   // GBK_TO_UNICODE[42068] := 16#F758;
   // GBK_TO_UNICODE[42069] := 16#9C54;
   // GBK_TO_UNICODE[42070] := 16#F759;
   // GBK_TO_UNICODE[42071] := 16#9C55;
   // GBK_TO_UNICODE[42072] := 16#F75A;
   // GBK_TO_UNICODE[42073] := 16#9C56;
   // GBK_TO_UNICODE[42074] := 16#F75B;
   // GBK_TO_UNICODE[42075] := 16#9C57;
   // GBK_TO_UNICODE[42076] := 16#F75C;
   // GBK_TO_UNICODE[42077] := 16#9C58;
   // GBK_TO_UNICODE[42078] := 16#F75D;
   // GBK_TO_UNICODE[42079] := 16#9C59;
   // GBK_TO_UNICODE[42080] := 16#F75E;
   // GBK_TO_UNICODE[42081] := 16#9C5A;
   // GBK_TO_UNICODE[42082] := 16#F75F;
   // GBK_TO_UNICODE[42083] := 16#9C5B;
   // GBK_TO_UNICODE[42084] := 16#F760;
   // GBK_TO_UNICODE[42085] := 16#9C5C;
   // GBK_TO_UNICODE[42086] := 16#F761;
   // GBK_TO_UNICODE[42087] := 16#9C5D;
   // GBK_TO_UNICODE[42088] := 16#F762;
   // GBK_TO_UNICODE[42089] := 16#9C5E;
   // GBK_TO_UNICODE[42090] := 16#F763;
   // GBK_TO_UNICODE[42091] := 16#9C5F;
   // GBK_TO_UNICODE[42092] := 16#F764;
   // GBK_TO_UNICODE[42093] := 16#9C60;
   // GBK_TO_UNICODE[42094] := 16#F765;
   // GBK_TO_UNICODE[42095] := 16#9C61;
   // GBK_TO_UNICODE[42096] := 16#F766;
   // GBK_TO_UNICODE[42097] := 16#9C62;
   // GBK_TO_UNICODE[42098] := 16#F767;
   // GBK_TO_UNICODE[42099] := 16#9C63;
   // GBK_TO_UNICODE[42100] := 16#F768;
   // GBK_TO_UNICODE[42101] := 16#9C64;
   // GBK_TO_UNICODE[42102] := 16#F769;
   // GBK_TO_UNICODE[42103] := 16#9C65;
   // GBK_TO_UNICODE[42104] := 16#F76A;
   // GBK_TO_UNICODE[42105] := 16#9C66;
   // GBK_TO_UNICODE[42106] := 16#F76B;
   // GBK_TO_UNICODE[42107] := 16#9C67;
   // GBK_TO_UNICODE[42108] := 16#F76C;
   // GBK_TO_UNICODE[42109] := 16#9C68;
   // GBK_TO_UNICODE[42110] := 16#F76D;
   // GBK_TO_UNICODE[42111] := 16#9C69;
   // GBK_TO_UNICODE[42112] := 16#F76E;
   // GBK_TO_UNICODE[42113] := 16#9C6A;
   // GBK_TO_UNICODE[42114] := 16#F76F;
   // GBK_TO_UNICODE[42115] := 16#9C6B;
   // GBK_TO_UNICODE[42116] := 16#F770;
   // GBK_TO_UNICODE[42117] := 16#9C6C;
   // GBK_TO_UNICODE[42118] := 16#F771;
   // GBK_TO_UNICODE[42119] := 16#9C6D;
   // GBK_TO_UNICODE[42120] := 16#F772;
   // GBK_TO_UNICODE[42121] := 16#9C6E;
   // GBK_TO_UNICODE[42122] := 16#F773;
   // GBK_TO_UNICODE[42123] := 16#9C6F;
   // GBK_TO_UNICODE[42124] := 16#F774;
   // GBK_TO_UNICODE[42125] := 16#9C70;
   // GBK_TO_UNICODE[42126] := 16#F775;
   // GBK_TO_UNICODE[42127] := 16#9C71;
   // GBK_TO_UNICODE[42128] := 16#F776;
   // GBK_TO_UNICODE[42129] := 16#9C72;
   // GBK_TO_UNICODE[42130] := 16#F777;
   // GBK_TO_UNICODE[42131] := 16#9C73;
   // GBK_TO_UNICODE[42132] := 16#F778;
   // GBK_TO_UNICODE[42133] := 16#9C74;
   // GBK_TO_UNICODE[42134] := 16#F779;
   // GBK_TO_UNICODE[42135] := 16#9C75;
   // GBK_TO_UNICODE[42136] := 16#F77A;
   // GBK_TO_UNICODE[42137] := 16#9C76;
   // GBK_TO_UNICODE[42138] := 16#F77B;
   // GBK_TO_UNICODE[42139] := 16#9C77;
   // GBK_TO_UNICODE[42140] := 16#F77C;
   // GBK_TO_UNICODE[42141] := 16#9C78;
   // GBK_TO_UNICODE[42142] := 16#F77D;
   // GBK_TO_UNICODE[42143] := 16#9C79;
   // GBK_TO_UNICODE[42144] := 16#F77E;
   // GBK_TO_UNICODE[42145] := 16#9C7A;
   // GBK_TO_UNICODE[42146] := 16#F780;
   // GBK_TO_UNICODE[42147] := 16#9C7B;
   // GBK_TO_UNICODE[42148] := 16#F781;
   // GBK_TO_UNICODE[42149] := 16#9C7D;
   // GBK_TO_UNICODE[42150] := 16#F782;
   // GBK_TO_UNICODE[42151] := 16#9C7E;
   // GBK_TO_UNICODE[42152] := 16#F783;
   // GBK_TO_UNICODE[42153] := 16#9C80;
   // GBK_TO_UNICODE[42154] := 16#F784;
   // GBK_TO_UNICODE[42155] := 16#9C83;
   // GBK_TO_UNICODE[42156] := 16#F785;
   // GBK_TO_UNICODE[42157] := 16#9C84;
   // GBK_TO_UNICODE[42158] := 16#F786;
   // GBK_TO_UNICODE[42159] := 16#9C89;
   // GBK_TO_UNICODE[42160] := 16#F787;
   // GBK_TO_UNICODE[42161] := 16#9C8A;
   // GBK_TO_UNICODE[42162] := 16#F788;
   // GBK_TO_UNICODE[42163] := 16#9C8C;
   // GBK_TO_UNICODE[42164] := 16#F789;
   // GBK_TO_UNICODE[42165] := 16#9C8F;
   // GBK_TO_UNICODE[42166] := 16#F78A;
   // GBK_TO_UNICODE[42167] := 16#9C93;
   // GBK_TO_UNICODE[42168] := 16#F78B;
   // GBK_TO_UNICODE[42169] := 16#9C96;
   // GBK_TO_UNICODE[42170] := 16#F78C;
   // GBK_TO_UNICODE[42171] := 16#9C97;
   // GBK_TO_UNICODE[42172] := 16#F78D;
   // GBK_TO_UNICODE[42173] := 16#9C98;
   // GBK_TO_UNICODE[42174] := 16#F78E;
   // GBK_TO_UNICODE[42175] := 16#9C99;
   // GBK_TO_UNICODE[42176] := 16#F78F;
   // GBK_TO_UNICODE[42177] := 16#9C9D;
   // GBK_TO_UNICODE[42178] := 16#F790;
   // GBK_TO_UNICODE[42179] := 16#9CAA;
   // GBK_TO_UNICODE[42180] := 16#F791;
   // GBK_TO_UNICODE[42181] := 16#9CAC;
   // GBK_TO_UNICODE[42182] := 16#F792;
   // GBK_TO_UNICODE[42183] := 16#9CAF;
   // GBK_TO_UNICODE[42184] := 16#F793;
   // GBK_TO_UNICODE[42185] := 16#9CB9;
   // GBK_TO_UNICODE[42186] := 16#F794;
   // GBK_TO_UNICODE[42187] := 16#9CBE;
   // GBK_TO_UNICODE[42188] := 16#F795;
   // GBK_TO_UNICODE[42189] := 16#9CBF;
   // GBK_TO_UNICODE[42190] := 16#F796;
   // GBK_TO_UNICODE[42191] := 16#9CC0;
   // GBK_TO_UNICODE[42192] := 16#F797;
   // GBK_TO_UNICODE[42193] := 16#9CC1;
   // GBK_TO_UNICODE[42194] := 16#F798;
   // GBK_TO_UNICODE[42195] := 16#9CC2;
   // GBK_TO_UNICODE[42196] := 16#F799;
   // GBK_TO_UNICODE[42197] := 16#9CC8;
   // GBK_TO_UNICODE[42198] := 16#F79A;
   // GBK_TO_UNICODE[42199] := 16#9CC9;
   // GBK_TO_UNICODE[42200] := 16#F79B;
   // GBK_TO_UNICODE[42201] := 16#9CD1;
   // GBK_TO_UNICODE[42202] := 16#F79C;
   // GBK_TO_UNICODE[42203] := 16#9CD2;
   // GBK_TO_UNICODE[42204] := 16#F79D;
   // GBK_TO_UNICODE[42205] := 16#9CDA;
   // GBK_TO_UNICODE[42206] := 16#F79E;
   // GBK_TO_UNICODE[42207] := 16#9CDB;
   // GBK_TO_UNICODE[42208] := 16#F79F;
   // GBK_TO_UNICODE[42209] := 16#9CE0;
   // GBK_TO_UNICODE[42210] := 16#F7A0;
   // GBK_TO_UNICODE[42211] := 16#9CE1;
   // GBK_TO_UNICODE[42212] := 16#F7A1;
   // GBK_TO_UNICODE[42213] := 16#9CCC;
   // GBK_TO_UNICODE[42214] := 16#F7A2;
   // GBK_TO_UNICODE[42215] := 16#9CCD;
   // GBK_TO_UNICODE[42216] := 16#F7A3;
   // GBK_TO_UNICODE[42217] := 16#9CCE;
   // GBK_TO_UNICODE[42218] := 16#F7A4;
   // GBK_TO_UNICODE[42219] := 16#9CCF;
   // GBK_TO_UNICODE[42220] := 16#F7A5;
   // GBK_TO_UNICODE[42221] := 16#9CD0;
   // GBK_TO_UNICODE[42222] := 16#F7A6;
   // GBK_TO_UNICODE[42223] := 16#9CD3;
   // GBK_TO_UNICODE[42224] := 16#F7A7;
   // GBK_TO_UNICODE[42225] := 16#9CD4;
   // GBK_TO_UNICODE[42226] := 16#F7A8;
   // GBK_TO_UNICODE[42227] := 16#9CD5;
   // GBK_TO_UNICODE[42228] := 16#F7A9;
   // GBK_TO_UNICODE[42229] := 16#9CD7;
   // GBK_TO_UNICODE[42230] := 16#F7AA;
   // GBK_TO_UNICODE[42231] := 16#9CD8;
   // GBK_TO_UNICODE[42232] := 16#F7AB;
   // GBK_TO_UNICODE[42233] := 16#9CD9;
   // GBK_TO_UNICODE[42234] := 16#F7AC;
   // GBK_TO_UNICODE[42235] := 16#9CDC;
   // GBK_TO_UNICODE[42236] := 16#F7AD;
   // GBK_TO_UNICODE[42237] := 16#9CDD;
   // GBK_TO_UNICODE[42238] := 16#F7AE;
   // GBK_TO_UNICODE[42239] := 16#9CDF;
   // GBK_TO_UNICODE[42240] := 16#F7AF;
   // GBK_TO_UNICODE[42241] := 16#9CE2;
   // GBK_TO_UNICODE[42242] := 16#F7B0;
   // GBK_TO_UNICODE[42243] := 16#977C;
   // GBK_TO_UNICODE[42244] := 16#F7B1;
   // GBK_TO_UNICODE[42245] := 16#9785;
   // GBK_TO_UNICODE[42246] := 16#F7B2;
   // GBK_TO_UNICODE[42247] := 16#9791;
   // GBK_TO_UNICODE[42248] := 16#F7B3;
   // GBK_TO_UNICODE[42249] := 16#9792;
   // GBK_TO_UNICODE[42250] := 16#F7B4;
   // GBK_TO_UNICODE[42251] := 16#9794;
   // GBK_TO_UNICODE[42252] := 16#F7B5;
   // GBK_TO_UNICODE[42253] := 16#97AF;
   // GBK_TO_UNICODE[42254] := 16#F7B6;
   // GBK_TO_UNICODE[42255] := 16#97AB;
   // GBK_TO_UNICODE[42256] := 16#F7B7;
   // GBK_TO_UNICODE[42257] := 16#97A3;
   // GBK_TO_UNICODE[42258] := 16#F7B8;
   // GBK_TO_UNICODE[42259] := 16#97B2;
   // GBK_TO_UNICODE[42260] := 16#F7B9;
   // GBK_TO_UNICODE[42261] := 16#97B4;
   // GBK_TO_UNICODE[42262] := 16#F7BA;
   // GBK_TO_UNICODE[42263] := 16#9AB1;
   // GBK_TO_UNICODE[42264] := 16#F7BB;
   // GBK_TO_UNICODE[42265] := 16#9AB0;
   // GBK_TO_UNICODE[42266] := 16#F7BC;
   // GBK_TO_UNICODE[42267] := 16#9AB7;
   // GBK_TO_UNICODE[42268] := 16#F7BD;
   // GBK_TO_UNICODE[42269] := 16#9E58;
   // GBK_TO_UNICODE[42270] := 16#F7BE;
   // GBK_TO_UNICODE[42271] := 16#9AB6;
   // GBK_TO_UNICODE[42272] := 16#F7BF;
   // GBK_TO_UNICODE[42273] := 16#9ABA;
   // GBK_TO_UNICODE[42274] := 16#F7C0;
   // GBK_TO_UNICODE[42275] := 16#9ABC;
   // GBK_TO_UNICODE[42276] := 16#F7C1;
   // GBK_TO_UNICODE[42277] := 16#9AC1;
   // GBK_TO_UNICODE[42278] := 16#F7C2;
   // GBK_TO_UNICODE[42279] := 16#9AC0;
   // GBK_TO_UNICODE[42280] := 16#F7C3;
   // GBK_TO_UNICODE[42281] := 16#9AC5;
   // GBK_TO_UNICODE[42282] := 16#F7C4;
   // GBK_TO_UNICODE[42283] := 16#9AC2;
   // GBK_TO_UNICODE[42284] := 16#F7C5;
   // GBK_TO_UNICODE[42285] := 16#9ACB;
   // GBK_TO_UNICODE[42286] := 16#F7C6;
   // GBK_TO_UNICODE[42287] := 16#9ACC;
   // GBK_TO_UNICODE[42288] := 16#F7C7;
   // GBK_TO_UNICODE[42289] := 16#9AD1;
   // GBK_TO_UNICODE[42290] := 16#F7C8;
   // GBK_TO_UNICODE[42291] := 16#9B45;
   // GBK_TO_UNICODE[42292] := 16#F7C9;
   // GBK_TO_UNICODE[42293] := 16#9B43;
   // GBK_TO_UNICODE[42294] := 16#F7CA;
   // GBK_TO_UNICODE[42295] := 16#9B47;
   // GBK_TO_UNICODE[42296] := 16#F7CB;
   // GBK_TO_UNICODE[42297] := 16#9B49;
   // GBK_TO_UNICODE[42298] := 16#F7CC;
   // GBK_TO_UNICODE[42299] := 16#9B48;
   // GBK_TO_UNICODE[42300] := 16#F7CD;
   // GBK_TO_UNICODE[42301] := 16#9B4D;
   // GBK_TO_UNICODE[42302] := 16#F7CE;
   // GBK_TO_UNICODE[42303] := 16#9B51;
   // GBK_TO_UNICODE[42304] := 16#F7CF;
   // GBK_TO_UNICODE[42305] := 16#98E8;
   // GBK_TO_UNICODE[42306] := 16#F7D0;
   // GBK_TO_UNICODE[42307] := 16#990D;
   // GBK_TO_UNICODE[42308] := 16#F7D1;
   // GBK_TO_UNICODE[42309] := 16#992E;
   // GBK_TO_UNICODE[42310] := 16#F7D2;
   // GBK_TO_UNICODE[42311] := 16#9955;
   // GBK_TO_UNICODE[42312] := 16#F7D3;
   // GBK_TO_UNICODE[42313] := 16#9954;
   // GBK_TO_UNICODE[42314] := 16#F7D4;
   // GBK_TO_UNICODE[42315] := 16#9ADF;
   // GBK_TO_UNICODE[42316] := 16#F7D5;
   // GBK_TO_UNICODE[42317] := 16#9AE1;
   // GBK_TO_UNICODE[42318] := 16#F7D6;
   // GBK_TO_UNICODE[42319] := 16#9AE6;
   // GBK_TO_UNICODE[42320] := 16#F7D7;
   // GBK_TO_UNICODE[42321] := 16#9AEF;
   // GBK_TO_UNICODE[42322] := 16#F7D8;
   // GBK_TO_UNICODE[42323] := 16#9AEB;
   // GBK_TO_UNICODE[42324] := 16#F7D9;
   // GBK_TO_UNICODE[42325] := 16#9AFB;
   // GBK_TO_UNICODE[42326] := 16#F7DA;
   // GBK_TO_UNICODE[42327] := 16#9AED;
   // GBK_TO_UNICODE[42328] := 16#F7DB;
   // GBK_TO_UNICODE[42329] := 16#9AF9;
   // GBK_TO_UNICODE[42330] := 16#F7DC;
   // GBK_TO_UNICODE[42331] := 16#9B08;
   // GBK_TO_UNICODE[42332] := 16#F7DD;
   // GBK_TO_UNICODE[42333] := 16#9B0F;
   // GBK_TO_UNICODE[42334] := 16#F7DE;
   // GBK_TO_UNICODE[42335] := 16#9B13;
   // GBK_TO_UNICODE[42336] := 16#F7DF;
   // GBK_TO_UNICODE[42337] := 16#9B1F;
   // GBK_TO_UNICODE[42338] := 16#F7E0;
   // GBK_TO_UNICODE[42339] := 16#9B23;
   // GBK_TO_UNICODE[42340] := 16#F7E1;
   // GBK_TO_UNICODE[42341] := 16#9EBD;
   // GBK_TO_UNICODE[42342] := 16#F7E2;
   // GBK_TO_UNICODE[42343] := 16#9EBE;
   // GBK_TO_UNICODE[42344] := 16#F7E3;
   // GBK_TO_UNICODE[42345] := 16#7E3B;
   // GBK_TO_UNICODE[42346] := 16#F7E4;
   // GBK_TO_UNICODE[42347] := 16#9E82;
   // GBK_TO_UNICODE[42348] := 16#F7E5;
   // GBK_TO_UNICODE[42349] := 16#9E87;
   // GBK_TO_UNICODE[42350] := 16#F7E6;
   // GBK_TO_UNICODE[42351] := 16#9E88;
   // GBK_TO_UNICODE[42352] := 16#F7E7;
   // GBK_TO_UNICODE[42353] := 16#9E8B;
   // GBK_TO_UNICODE[42354] := 16#F7E8;
   // GBK_TO_UNICODE[42355] := 16#9E92;
   // GBK_TO_UNICODE[42356] := 16#F7E9;
   // GBK_TO_UNICODE[42357] := 16#93D6;
   // GBK_TO_UNICODE[42358] := 16#F7EA;
   // GBK_TO_UNICODE[42359] := 16#9E9D;
   // GBK_TO_UNICODE[42360] := 16#F7EB;
   // GBK_TO_UNICODE[42361] := 16#9E9F;
   // GBK_TO_UNICODE[42362] := 16#F7EC;
   // GBK_TO_UNICODE[42363] := 16#9EDB;
   // GBK_TO_UNICODE[42364] := 16#F7ED;
   // GBK_TO_UNICODE[42365] := 16#9EDC;
   // GBK_TO_UNICODE[42366] := 16#F7EE;
   // GBK_TO_UNICODE[42367] := 16#9EDD;
   // GBK_TO_UNICODE[42368] := 16#F7EF;
   // GBK_TO_UNICODE[42369] := 16#9EE0;
   // GBK_TO_UNICODE[42370] := 16#F7F0;
   // GBK_TO_UNICODE[42371] := 16#9EDF;
   // GBK_TO_UNICODE[42372] := 16#F7F1;
   // GBK_TO_UNICODE[42373] := 16#9EE2;
   // GBK_TO_UNICODE[42374] := 16#F7F2;
   // GBK_TO_UNICODE[42375] := 16#9EE9;
   // GBK_TO_UNICODE[42376] := 16#F7F3;
   // GBK_TO_UNICODE[42377] := 16#9EE7;
   // GBK_TO_UNICODE[42378] := 16#F7F4;
   // GBK_TO_UNICODE[42379] := 16#9EE5;
   // GBK_TO_UNICODE[42380] := 16#F7F5;
   // GBK_TO_UNICODE[42381] := 16#9EEA;
   // GBK_TO_UNICODE[42382] := 16#F7F6;
   // GBK_TO_UNICODE[42383] := 16#9EEF;
   // GBK_TO_UNICODE[42384] := 16#F7F7;
   // GBK_TO_UNICODE[42385] := 16#9F22;
   // GBK_TO_UNICODE[42386] := 16#F7F8;
   // GBK_TO_UNICODE[42387] := 16#9F2C;
   // GBK_TO_UNICODE[42388] := 16#F7F9;
   // GBK_TO_UNICODE[42389] := 16#9F2F;
   // GBK_TO_UNICODE[42390] := 16#F7FA;
   // GBK_TO_UNICODE[42391] := 16#9F39;
   // GBK_TO_UNICODE[42392] := 16#F7FB;
   // GBK_TO_UNICODE[42393] := 16#9F37;
   // GBK_TO_UNICODE[42394] := 16#F7FC;
   // GBK_TO_UNICODE[42395] := 16#9F3D;
   // GBK_TO_UNICODE[42396] := 16#F7FD;
   // GBK_TO_UNICODE[42397] := 16#9F3E;
   // GBK_TO_UNICODE[42398] := 16#F7FE;
   // GBK_TO_UNICODE[42399] := 16#9F44;
   // GBK_TO_UNICODE[42400] := 16#F840;
   // GBK_TO_UNICODE[42401] := 16#9CE3;
   // GBK_TO_UNICODE[42402] := 16#F841;
   // GBK_TO_UNICODE[42403] := 16#9CE4;
   // GBK_TO_UNICODE[42404] := 16#F842;
   // GBK_TO_UNICODE[42405] := 16#9CE5;
   // GBK_TO_UNICODE[42406] := 16#F843;
   // GBK_TO_UNICODE[42407] := 16#9CE6;
   // GBK_TO_UNICODE[42408] := 16#F844;
   // GBK_TO_UNICODE[42409] := 16#9CE7;
   // GBK_TO_UNICODE[42410] := 16#F845;
   // GBK_TO_UNICODE[42411] := 16#9CE8;
   // GBK_TO_UNICODE[42412] := 16#F846;
   // GBK_TO_UNICODE[42413] := 16#9CE9;
   // GBK_TO_UNICODE[42414] := 16#F847;
   // GBK_TO_UNICODE[42415] := 16#9CEA;
   // GBK_TO_UNICODE[42416] := 16#F848;
   // GBK_TO_UNICODE[42417] := 16#9CEB;
   // GBK_TO_UNICODE[42418] := 16#F849;
   // GBK_TO_UNICODE[42419] := 16#9CEC;
   // GBK_TO_UNICODE[42420] := 16#F84A;
   // GBK_TO_UNICODE[42421] := 16#9CED;
   // GBK_TO_UNICODE[42422] := 16#F84B;
   // GBK_TO_UNICODE[42423] := 16#9CEE;
   // GBK_TO_UNICODE[42424] := 16#F84C;
   // GBK_TO_UNICODE[42425] := 16#9CEF;
   // GBK_TO_UNICODE[42426] := 16#F84D;
   // GBK_TO_UNICODE[42427] := 16#9CF0;
   // GBK_TO_UNICODE[42428] := 16#F84E;
   // GBK_TO_UNICODE[42429] := 16#9CF1;
   // GBK_TO_UNICODE[42430] := 16#F84F;
   // GBK_TO_UNICODE[42431] := 16#9CF2;
   // GBK_TO_UNICODE[42432] := 16#F850;
   // GBK_TO_UNICODE[42433] := 16#9CF3;
   // GBK_TO_UNICODE[42434] := 16#F851;
   // GBK_TO_UNICODE[42435] := 16#9CF4;
   // GBK_TO_UNICODE[42436] := 16#F852;
   // GBK_TO_UNICODE[42437] := 16#9CF5;
   // GBK_TO_UNICODE[42438] := 16#F853;
   // GBK_TO_UNICODE[42439] := 16#9CF6;
   // GBK_TO_UNICODE[42440] := 16#F854;
   // GBK_TO_UNICODE[42441] := 16#9CF7;
   // GBK_TO_UNICODE[42442] := 16#F855;
   // GBK_TO_UNICODE[42443] := 16#9CF8;
   // GBK_TO_UNICODE[42444] := 16#F856;
   // GBK_TO_UNICODE[42445] := 16#9CF9;
   // GBK_TO_UNICODE[42446] := 16#F857;
   // GBK_TO_UNICODE[42447] := 16#9CFA;
   // GBK_TO_UNICODE[42448] := 16#F858;
   // GBK_TO_UNICODE[42449] := 16#9CFB;
   // GBK_TO_UNICODE[42450] := 16#F859;
   // GBK_TO_UNICODE[42451] := 16#9CFC;
   // GBK_TO_UNICODE[42452] := 16#F85A;
   // GBK_TO_UNICODE[42453] := 16#9CFD;
   // GBK_TO_UNICODE[42454] := 16#F85B;
   // GBK_TO_UNICODE[42455] := 16#9CFE;
   // GBK_TO_UNICODE[42456] := 16#F85C;
   // GBK_TO_UNICODE[42457] := 16#9CFF;
   // GBK_TO_UNICODE[42458] := 16#F85D;
   // GBK_TO_UNICODE[42459] := 16#9D00;
   // GBK_TO_UNICODE[42460] := 16#F85E;
   // GBK_TO_UNICODE[42461] := 16#9D01;
   // GBK_TO_UNICODE[42462] := 16#F85F;
   // GBK_TO_UNICODE[42463] := 16#9D02;
   // GBK_TO_UNICODE[42464] := 16#F860;
   // GBK_TO_UNICODE[42465] := 16#9D03;
   // GBK_TO_UNICODE[42466] := 16#F861;
   // GBK_TO_UNICODE[42467] := 16#9D04;
   // GBK_TO_UNICODE[42468] := 16#F862;
   // GBK_TO_UNICODE[42469] := 16#9D05;
   // GBK_TO_UNICODE[42470] := 16#F863;
   // GBK_TO_UNICODE[42471] := 16#9D06;
   // GBK_TO_UNICODE[42472] := 16#F864;
   // GBK_TO_UNICODE[42473] := 16#9D07;
   // GBK_TO_UNICODE[42474] := 16#F865;
   // GBK_TO_UNICODE[42475] := 16#9D08;
   // GBK_TO_UNICODE[42476] := 16#F866;
   // GBK_TO_UNICODE[42477] := 16#9D09;
   // GBK_TO_UNICODE[42478] := 16#F867;
   // GBK_TO_UNICODE[42479] := 16#9D0A;
   // GBK_TO_UNICODE[42480] := 16#F868;
   // GBK_TO_UNICODE[42481] := 16#9D0B;
   // GBK_TO_UNICODE[42482] := 16#F869;
   // GBK_TO_UNICODE[42483] := 16#9D0C;
   // GBK_TO_UNICODE[42484] := 16#F86A;
   // GBK_TO_UNICODE[42485] := 16#9D0D;
   // GBK_TO_UNICODE[42486] := 16#F86B;
   // GBK_TO_UNICODE[42487] := 16#9D0E;
   // GBK_TO_UNICODE[42488] := 16#F86C;
   // GBK_TO_UNICODE[42489] := 16#9D0F;
   // GBK_TO_UNICODE[42490] := 16#F86D;
   // GBK_TO_UNICODE[42491] := 16#9D10;
   // GBK_TO_UNICODE[42492] := 16#F86E;
   // GBK_TO_UNICODE[42493] := 16#9D11;
   // GBK_TO_UNICODE[42494] := 16#F86F;
   // GBK_TO_UNICODE[42495] := 16#9D12;
   // GBK_TO_UNICODE[42496] := 16#F870;
   // GBK_TO_UNICODE[42497] := 16#9D13;
   // GBK_TO_UNICODE[42498] := 16#F871;
   // GBK_TO_UNICODE[42499] := 16#9D14;
   // GBK_TO_UNICODE[42500] := 16#F872;
   // GBK_TO_UNICODE[42501] := 16#9D15;
   // GBK_TO_UNICODE[42502] := 16#F873;
   // GBK_TO_UNICODE[42503] := 16#9D16;
   // GBK_TO_UNICODE[42504] := 16#F874;
   // GBK_TO_UNICODE[42505] := 16#9D17;
   // GBK_TO_UNICODE[42506] := 16#F875;
   // GBK_TO_UNICODE[42507] := 16#9D18;
   // GBK_TO_UNICODE[42508] := 16#F876;
   // GBK_TO_UNICODE[42509] := 16#9D19;
   // GBK_TO_UNICODE[42510] := 16#F877;
   // GBK_TO_UNICODE[42511] := 16#9D1A;
   // GBK_TO_UNICODE[42512] := 16#F878;
   // GBK_TO_UNICODE[42513] := 16#9D1B;
   // GBK_TO_UNICODE[42514] := 16#F879;
   // GBK_TO_UNICODE[42515] := 16#9D1C;
   // GBK_TO_UNICODE[42516] := 16#F87A;
   // GBK_TO_UNICODE[42517] := 16#9D1D;
   // GBK_TO_UNICODE[42518] := 16#F87B;
   // GBK_TO_UNICODE[42519] := 16#9D1E;
   // GBK_TO_UNICODE[42520] := 16#F87C;
   // GBK_TO_UNICODE[42521] := 16#9D1F;
   // GBK_TO_UNICODE[42522] := 16#F87D;
   // GBK_TO_UNICODE[42523] := 16#9D20;
   // GBK_TO_UNICODE[42524] := 16#F87E;
   // GBK_TO_UNICODE[42525] := 16#9D21;
   // GBK_TO_UNICODE[42526] := 16#F880;
   // GBK_TO_UNICODE[42527] := 16#9D22;
   // GBK_TO_UNICODE[42528] := 16#F881;
   // GBK_TO_UNICODE[42529] := 16#9D23;
   // GBK_TO_UNICODE[42530] := 16#F882;
   // GBK_TO_UNICODE[42531] := 16#9D24;
   // GBK_TO_UNICODE[42532] := 16#F883;
   // GBK_TO_UNICODE[42533] := 16#9D25;
   // GBK_TO_UNICODE[42534] := 16#F884;
   // GBK_TO_UNICODE[42535] := 16#9D26;
   // GBK_TO_UNICODE[42536] := 16#F885;
   // GBK_TO_UNICODE[42537] := 16#9D27;
   // GBK_TO_UNICODE[42538] := 16#F886;
   // GBK_TO_UNICODE[42539] := 16#9D28;
   // GBK_TO_UNICODE[42540] := 16#F887;
   // GBK_TO_UNICODE[42541] := 16#9D29;
   // GBK_TO_UNICODE[42542] := 16#F888;
   // GBK_TO_UNICODE[42543] := 16#9D2A;
   // GBK_TO_UNICODE[42544] := 16#F889;
   // GBK_TO_UNICODE[42545] := 16#9D2B;
   // GBK_TO_UNICODE[42546] := 16#F88A;
   // GBK_TO_UNICODE[42547] := 16#9D2C;
   // GBK_TO_UNICODE[42548] := 16#F88B;
   // GBK_TO_UNICODE[42549] := 16#9D2D;
   // GBK_TO_UNICODE[42550] := 16#F88C;
   // GBK_TO_UNICODE[42551] := 16#9D2E;
   // GBK_TO_UNICODE[42552] := 16#F88D;
   // GBK_TO_UNICODE[42553] := 16#9D2F;
   // GBK_TO_UNICODE[42554] := 16#F88E;
   // GBK_TO_UNICODE[42555] := 16#9D30;
   // GBK_TO_UNICODE[42556] := 16#F88F;
   // GBK_TO_UNICODE[42557] := 16#9D31;
   // GBK_TO_UNICODE[42558] := 16#F890;
   // GBK_TO_UNICODE[42559] := 16#9D32;
   // GBK_TO_UNICODE[42560] := 16#F891;
   // GBK_TO_UNICODE[42561] := 16#9D33;
   // GBK_TO_UNICODE[42562] := 16#F892;
   // GBK_TO_UNICODE[42563] := 16#9D34;
   // GBK_TO_UNICODE[42564] := 16#F893;
   // GBK_TO_UNICODE[42565] := 16#9D35;
   // GBK_TO_UNICODE[42566] := 16#F894;
   // GBK_TO_UNICODE[42567] := 16#9D36;
   // GBK_TO_UNICODE[42568] := 16#F895;
   // GBK_TO_UNICODE[42569] := 16#9D37;
   // GBK_TO_UNICODE[42570] := 16#F896;
   // GBK_TO_UNICODE[42571] := 16#9D38;
   // GBK_TO_UNICODE[42572] := 16#F897;
   // GBK_TO_UNICODE[42573] := 16#9D39;
   // GBK_TO_UNICODE[42574] := 16#F898;
   // GBK_TO_UNICODE[42575] := 16#9D3A;
   // GBK_TO_UNICODE[42576] := 16#F899;
   // GBK_TO_UNICODE[42577] := 16#9D3B;
   // GBK_TO_UNICODE[42578] := 16#F89A;
   // GBK_TO_UNICODE[42579] := 16#9D3C;
   // GBK_TO_UNICODE[42580] := 16#F89B;
   // GBK_TO_UNICODE[42581] := 16#9D3D;
   // GBK_TO_UNICODE[42582] := 16#F89C;
   // GBK_TO_UNICODE[42583] := 16#9D3E;
   // GBK_TO_UNICODE[42584] := 16#F89D;
   // GBK_TO_UNICODE[42585] := 16#9D3F;
   // GBK_TO_UNICODE[42586] := 16#F89E;
   // GBK_TO_UNICODE[42587] := 16#9D40;
   // GBK_TO_UNICODE[42588] := 16#F89F;
   // GBK_TO_UNICODE[42589] := 16#9D41;
   // GBK_TO_UNICODE[42590] := 16#F8A0;
   // GBK_TO_UNICODE[42591] := 16#9D42;
   // GBK_TO_UNICODE[42592] := 16#F940;
   // GBK_TO_UNICODE[42593] := 16#9D43;
   // GBK_TO_UNICODE[42594] := 16#F941;
   // GBK_TO_UNICODE[42595] := 16#9D44;
   // GBK_TO_UNICODE[42596] := 16#F942;
   // GBK_TO_UNICODE[42597] := 16#9D45;
   // GBK_TO_UNICODE[42598] := 16#F943;
   // GBK_TO_UNICODE[42599] := 16#9D46;
   // GBK_TO_UNICODE[42600] := 16#F944;
   // GBK_TO_UNICODE[42601] := 16#9D47;
   // GBK_TO_UNICODE[42602] := 16#F945;
   // GBK_TO_UNICODE[42603] := 16#9D48;
   // GBK_TO_UNICODE[42604] := 16#F946;
   // GBK_TO_UNICODE[42605] := 16#9D49;
   // GBK_TO_UNICODE[42606] := 16#F947;
   // GBK_TO_UNICODE[42607] := 16#9D4A;
   // GBK_TO_UNICODE[42608] := 16#F948;
   // GBK_TO_UNICODE[42609] := 16#9D4B;
   // GBK_TO_UNICODE[42610] := 16#F949;
   // GBK_TO_UNICODE[42611] := 16#9D4C;
   // GBK_TO_UNICODE[42612] := 16#F94A;
   // GBK_TO_UNICODE[42613] := 16#9D4D;
   // GBK_TO_UNICODE[42614] := 16#F94B;
   // GBK_TO_UNICODE[42615] := 16#9D4E;
   // GBK_TO_UNICODE[42616] := 16#F94C;
   // GBK_TO_UNICODE[42617] := 16#9D4F;
   // GBK_TO_UNICODE[42618] := 16#F94D;
   // GBK_TO_UNICODE[42619] := 16#9D50;
   // GBK_TO_UNICODE[42620] := 16#F94E;
   // GBK_TO_UNICODE[42621] := 16#9D51;
   // GBK_TO_UNICODE[42622] := 16#F94F;
   // GBK_TO_UNICODE[42623] := 16#9D52;
   // GBK_TO_UNICODE[42624] := 16#F950;
   // GBK_TO_UNICODE[42625] := 16#9D53;
   // GBK_TO_UNICODE[42626] := 16#F951;
   // GBK_TO_UNICODE[42627] := 16#9D54;
   // GBK_TO_UNICODE[42628] := 16#F952;
   // GBK_TO_UNICODE[42629] := 16#9D55;
   // GBK_TO_UNICODE[42630] := 16#F953;
   // GBK_TO_UNICODE[42631] := 16#9D56;
   // GBK_TO_UNICODE[42632] := 16#F954;
   // GBK_TO_UNICODE[42633] := 16#9D57;
   // GBK_TO_UNICODE[42634] := 16#F955;
   // GBK_TO_UNICODE[42635] := 16#9D58;
   // GBK_TO_UNICODE[42636] := 16#F956;
   // GBK_TO_UNICODE[42637] := 16#9D59;
   // GBK_TO_UNICODE[42638] := 16#F957;
   // GBK_TO_UNICODE[42639] := 16#9D5A;
   // GBK_TO_UNICODE[42640] := 16#F958;
   // GBK_TO_UNICODE[42641] := 16#9D5B;
   // GBK_TO_UNICODE[42642] := 16#F959;
   // GBK_TO_UNICODE[42643] := 16#9D5C;
   // GBK_TO_UNICODE[42644] := 16#F95A;
   // GBK_TO_UNICODE[42645] := 16#9D5D;
   // GBK_TO_UNICODE[42646] := 16#F95B;
   // GBK_TO_UNICODE[42647] := 16#9D5E;
   // GBK_TO_UNICODE[42648] := 16#F95C;
   // GBK_TO_UNICODE[42649] := 16#9D5F;
   // GBK_TO_UNICODE[42650] := 16#F95D;
   // GBK_TO_UNICODE[42651] := 16#9D60;
   // GBK_TO_UNICODE[42652] := 16#F95E;
   // GBK_TO_UNICODE[42653] := 16#9D61;
   // GBK_TO_UNICODE[42654] := 16#F95F;
   // GBK_TO_UNICODE[42655] := 16#9D62;
   // GBK_TO_UNICODE[42656] := 16#F960;
   // GBK_TO_UNICODE[42657] := 16#9D63;
   // GBK_TO_UNICODE[42658] := 16#F961;
   // GBK_TO_UNICODE[42659] := 16#9D64;
   // GBK_TO_UNICODE[42660] := 16#F962;
   // GBK_TO_UNICODE[42661] := 16#9D65;
   // GBK_TO_UNICODE[42662] := 16#F963;
   // GBK_TO_UNICODE[42663] := 16#9D66;
   // GBK_TO_UNICODE[42664] := 16#F964;
   // GBK_TO_UNICODE[42665] := 16#9D67;
   // GBK_TO_UNICODE[42666] := 16#F965;
   // GBK_TO_UNICODE[42667] := 16#9D68;
   // GBK_TO_UNICODE[42668] := 16#F966;
   // GBK_TO_UNICODE[42669] := 16#9D69;
   // GBK_TO_UNICODE[42670] := 16#F967;
   // GBK_TO_UNICODE[42671] := 16#9D6A;
   // GBK_TO_UNICODE[42672] := 16#F968;
   // GBK_TO_UNICODE[42673] := 16#9D6B;
   // GBK_TO_UNICODE[42674] := 16#F969;
   // GBK_TO_UNICODE[42675] := 16#9D6C;
   // GBK_TO_UNICODE[42676] := 16#F96A;
   // GBK_TO_UNICODE[42677] := 16#9D6D;
   // GBK_TO_UNICODE[42678] := 16#F96B;
   // GBK_TO_UNICODE[42679] := 16#9D6E;
   // GBK_TO_UNICODE[42680] := 16#F96C;
   // GBK_TO_UNICODE[42681] := 16#9D6F;
   // GBK_TO_UNICODE[42682] := 16#F96D;
   // GBK_TO_UNICODE[42683] := 16#9D70;
   // GBK_TO_UNICODE[42684] := 16#F96E;
   // GBK_TO_UNICODE[42685] := 16#9D71;
   // GBK_TO_UNICODE[42686] := 16#F96F;
   // GBK_TO_UNICODE[42687] := 16#9D72;
   // GBK_TO_UNICODE[42688] := 16#F970;
   // GBK_TO_UNICODE[42689] := 16#9D73;
   // GBK_TO_UNICODE[42690] := 16#F971;
   // GBK_TO_UNICODE[42691] := 16#9D74;
   // GBK_TO_UNICODE[42692] := 16#F972;
   // GBK_TO_UNICODE[42693] := 16#9D75;
   // GBK_TO_UNICODE[42694] := 16#F973;
   // GBK_TO_UNICODE[42695] := 16#9D76;
   // GBK_TO_UNICODE[42696] := 16#F974;
   // GBK_TO_UNICODE[42697] := 16#9D77;
   // GBK_TO_UNICODE[42698] := 16#F975;
   // GBK_TO_UNICODE[42699] := 16#9D78;
   // GBK_TO_UNICODE[42700] := 16#F976;
   // GBK_TO_UNICODE[42701] := 16#9D79;
   // GBK_TO_UNICODE[42702] := 16#F977;
   // GBK_TO_UNICODE[42703] := 16#9D7A;
   // GBK_TO_UNICODE[42704] := 16#F978;
   // GBK_TO_UNICODE[42705] := 16#9D7B;
   // GBK_TO_UNICODE[42706] := 16#F979;
   // GBK_TO_UNICODE[42707] := 16#9D7C;
   // GBK_TO_UNICODE[42708] := 16#F97A;
   // GBK_TO_UNICODE[42709] := 16#9D7D;
   // GBK_TO_UNICODE[42710] := 16#F97B;
   // GBK_TO_UNICODE[42711] := 16#9D7E;
   // GBK_TO_UNICODE[42712] := 16#F97C;
   // GBK_TO_UNICODE[42713] := 16#9D7F;
   // GBK_TO_UNICODE[42714] := 16#F97D;
   // GBK_TO_UNICODE[42715] := 16#9D80;
   // GBK_TO_UNICODE[42716] := 16#F97E;
   // GBK_TO_UNICODE[42717] := 16#9D81;
   // GBK_TO_UNICODE[42718] := 16#F980;
   // GBK_TO_UNICODE[42719] := 16#9D82;
   // GBK_TO_UNICODE[42720] := 16#F981;
   // GBK_TO_UNICODE[42721] := 16#9D83;
   // GBK_TO_UNICODE[42722] := 16#F982;
   // GBK_TO_UNICODE[42723] := 16#9D84;
   // GBK_TO_UNICODE[42724] := 16#F983;
   // GBK_TO_UNICODE[42725] := 16#9D85;
   // GBK_TO_UNICODE[42726] := 16#F984;
   // GBK_TO_UNICODE[42727] := 16#9D86;
   // GBK_TO_UNICODE[42728] := 16#F985;
   // GBK_TO_UNICODE[42729] := 16#9D87;
   // GBK_TO_UNICODE[42730] := 16#F986;
   // GBK_TO_UNICODE[42731] := 16#9D88;
   // GBK_TO_UNICODE[42732] := 16#F987;
   // GBK_TO_UNICODE[42733] := 16#9D89;
   // GBK_TO_UNICODE[42734] := 16#F988;
   // GBK_TO_UNICODE[42735] := 16#9D8A;
   // GBK_TO_UNICODE[42736] := 16#F989;
   // GBK_TO_UNICODE[42737] := 16#9D8B;
   // GBK_TO_UNICODE[42738] := 16#F98A;
   // GBK_TO_UNICODE[42739] := 16#9D8C;
   // GBK_TO_UNICODE[42740] := 16#F98B;
   // GBK_TO_UNICODE[42741] := 16#9D8D;
   // GBK_TO_UNICODE[42742] := 16#F98C;
   // GBK_TO_UNICODE[42743] := 16#9D8E;
   // GBK_TO_UNICODE[42744] := 16#F98D;
   // GBK_TO_UNICODE[42745] := 16#9D8F;
   // GBK_TO_UNICODE[42746] := 16#F98E;
   // GBK_TO_UNICODE[42747] := 16#9D90;
   // GBK_TO_UNICODE[42748] := 16#F98F;
   // GBK_TO_UNICODE[42749] := 16#9D91;
   // GBK_TO_UNICODE[42750] := 16#F990;
   // GBK_TO_UNICODE[42751] := 16#9D92;
   // GBK_TO_UNICODE[42752] := 16#F991;
   // GBK_TO_UNICODE[42753] := 16#9D93;
   // GBK_TO_UNICODE[42754] := 16#F992;
   // GBK_TO_UNICODE[42755] := 16#9D94;
   // GBK_TO_UNICODE[42756] := 16#F993;
   // GBK_TO_UNICODE[42757] := 16#9D95;
   // GBK_TO_UNICODE[42758] := 16#F994;
   // GBK_TO_UNICODE[42759] := 16#9D96;
   // GBK_TO_UNICODE[42760] := 16#F995;
   // GBK_TO_UNICODE[42761] := 16#9D97;
   // GBK_TO_UNICODE[42762] := 16#F996;
   // GBK_TO_UNICODE[42763] := 16#9D98;
   // GBK_TO_UNICODE[42764] := 16#F997;
   // GBK_TO_UNICODE[42765] := 16#9D99;
   // GBK_TO_UNICODE[42766] := 16#F998;
   // GBK_TO_UNICODE[42767] := 16#9D9A;
   // GBK_TO_UNICODE[42768] := 16#F999;
   // GBK_TO_UNICODE[42769] := 16#9D9B;
   // GBK_TO_UNICODE[42770] := 16#F99A;
   // GBK_TO_UNICODE[42771] := 16#9D9C;
   // GBK_TO_UNICODE[42772] := 16#F99B;
   // GBK_TO_UNICODE[42773] := 16#9D9D;
   // GBK_TO_UNICODE[42774] := 16#F99C;
   // GBK_TO_UNICODE[42775] := 16#9D9E;
   // GBK_TO_UNICODE[42776] := 16#F99D;
   // GBK_TO_UNICODE[42777] := 16#9D9F;
   // GBK_TO_UNICODE[42778] := 16#F99E;
   // GBK_TO_UNICODE[42779] := 16#9DA0;
   // GBK_TO_UNICODE[42780] := 16#F99F;
   // GBK_TO_UNICODE[42781] := 16#9DA1;
   // GBK_TO_UNICODE[42782] := 16#F9A0;
   // GBK_TO_UNICODE[42783] := 16#9DA2;
   // GBK_TO_UNICODE[42784] := 16#FA40;
   // GBK_TO_UNICODE[42785] := 16#9DA3;
   // GBK_TO_UNICODE[42786] := 16#FA41;
   // GBK_TO_UNICODE[42787] := 16#9DA4;
   // GBK_TO_UNICODE[42788] := 16#FA42;
   // GBK_TO_UNICODE[42789] := 16#9DA5;
   // GBK_TO_UNICODE[42790] := 16#FA43;
   // GBK_TO_UNICODE[42791] := 16#9DA6;
   // GBK_TO_UNICODE[42792] := 16#FA44;
   // GBK_TO_UNICODE[42793] := 16#9DA7;
   // GBK_TO_UNICODE[42794] := 16#FA45;
   // GBK_TO_UNICODE[42795] := 16#9DA8;
   // GBK_TO_UNICODE[42796] := 16#FA46;
   // GBK_TO_UNICODE[42797] := 16#9DA9;
   // GBK_TO_UNICODE[42798] := 16#FA47;
   // GBK_TO_UNICODE[42799] := 16#9DAA;
   // GBK_TO_UNICODE[42800] := 16#FA48;
   // GBK_TO_UNICODE[42801] := 16#9DAB;
   // GBK_TO_UNICODE[42802] := 16#FA49;
   // GBK_TO_UNICODE[42803] := 16#9DAC;
   // GBK_TO_UNICODE[42804] := 16#FA4A;
   // GBK_TO_UNICODE[42805] := 16#9DAD;
   // GBK_TO_UNICODE[42806] := 16#FA4B;
   // GBK_TO_UNICODE[42807] := 16#9DAE;
   // GBK_TO_UNICODE[42808] := 16#FA4C;
   // GBK_TO_UNICODE[42809] := 16#9DAF;
   // GBK_TO_UNICODE[42810] := 16#FA4D;
   // GBK_TO_UNICODE[42811] := 16#9DB0;
   // GBK_TO_UNICODE[42812] := 16#FA4E;
   // GBK_TO_UNICODE[42813] := 16#9DB1;
   // GBK_TO_UNICODE[42814] := 16#FA4F;
   // GBK_TO_UNICODE[42815] := 16#9DB2;
   // GBK_TO_UNICODE[42816] := 16#FA50;
   // GBK_TO_UNICODE[42817] := 16#9DB3;
   // GBK_TO_UNICODE[42818] := 16#FA51;
   // GBK_TO_UNICODE[42819] := 16#9DB4;
   // GBK_TO_UNICODE[42820] := 16#FA52;
   // GBK_TO_UNICODE[42821] := 16#9DB5;
   // GBK_TO_UNICODE[42822] := 16#FA53;
   // GBK_TO_UNICODE[42823] := 16#9DB6;
   // GBK_TO_UNICODE[42824] := 16#FA54;
   // GBK_TO_UNICODE[42825] := 16#9DB7;
   // GBK_TO_UNICODE[42826] := 16#FA55;
   // GBK_TO_UNICODE[42827] := 16#9DB8;
   // GBK_TO_UNICODE[42828] := 16#FA56;
   // GBK_TO_UNICODE[42829] := 16#9DB9;
   // GBK_TO_UNICODE[42830] := 16#FA57;
   // GBK_TO_UNICODE[42831] := 16#9DBA;
   // GBK_TO_UNICODE[42832] := 16#FA58;
   // GBK_TO_UNICODE[42833] := 16#9DBB;
   // GBK_TO_UNICODE[42834] := 16#FA59;
   // GBK_TO_UNICODE[42835] := 16#9DBC;
   // GBK_TO_UNICODE[42836] := 16#FA5A;
   // GBK_TO_UNICODE[42837] := 16#9DBD;
   // GBK_TO_UNICODE[42838] := 16#FA5B;
   // GBK_TO_UNICODE[42839] := 16#9DBE;
   // GBK_TO_UNICODE[42840] := 16#FA5C;
   // GBK_TO_UNICODE[42841] := 16#9DBF;
   // GBK_TO_UNICODE[42842] := 16#FA5D;
   // GBK_TO_UNICODE[42843] := 16#9DC0;
   // GBK_TO_UNICODE[42844] := 16#FA5E;
   // GBK_TO_UNICODE[42845] := 16#9DC1;
   // GBK_TO_UNICODE[42846] := 16#FA5F;
   // GBK_TO_UNICODE[42847] := 16#9DC2;
   // GBK_TO_UNICODE[42848] := 16#FA60;
   // GBK_TO_UNICODE[42849] := 16#9DC3;
   // GBK_TO_UNICODE[42850] := 16#FA61;
   // GBK_TO_UNICODE[42851] := 16#9DC4;
   // GBK_TO_UNICODE[42852] := 16#FA62;
   // GBK_TO_UNICODE[42853] := 16#9DC5;
   // GBK_TO_UNICODE[42854] := 16#FA63;
   // GBK_TO_UNICODE[42855] := 16#9DC6;
   // GBK_TO_UNICODE[42856] := 16#FA64;
   // GBK_TO_UNICODE[42857] := 16#9DC7;
   // GBK_TO_UNICODE[42858] := 16#FA65;
   // GBK_TO_UNICODE[42859] := 16#9DC8;
   // GBK_TO_UNICODE[42860] := 16#FA66;
   // GBK_TO_UNICODE[42861] := 16#9DC9;
   // GBK_TO_UNICODE[42862] := 16#FA67;
   // GBK_TO_UNICODE[42863] := 16#9DCA;
   // GBK_TO_UNICODE[42864] := 16#FA68;
   // GBK_TO_UNICODE[42865] := 16#9DCB;
   // GBK_TO_UNICODE[42866] := 16#FA69;
   // GBK_TO_UNICODE[42867] := 16#9DCC;
   // GBK_TO_UNICODE[42868] := 16#FA6A;
   // GBK_TO_UNICODE[42869] := 16#9DCD;
   // GBK_TO_UNICODE[42870] := 16#FA6B;
   // GBK_TO_UNICODE[42871] := 16#9DCE;
   // GBK_TO_UNICODE[42872] := 16#FA6C;
   // GBK_TO_UNICODE[42873] := 16#9DCF;
   // GBK_TO_UNICODE[42874] := 16#FA6D;
   // GBK_TO_UNICODE[42875] := 16#9DD0;
   // GBK_TO_UNICODE[42876] := 16#FA6E;
   // GBK_TO_UNICODE[42877] := 16#9DD1;
   // GBK_TO_UNICODE[42878] := 16#FA6F;
   // GBK_TO_UNICODE[42879] := 16#9DD2;
   // GBK_TO_UNICODE[42880] := 16#FA70;
   // GBK_TO_UNICODE[42881] := 16#9DD3;
   // GBK_TO_UNICODE[42882] := 16#FA71;
   // GBK_TO_UNICODE[42883] := 16#9DD4;
   // GBK_TO_UNICODE[42884] := 16#FA72;
   // GBK_TO_UNICODE[42885] := 16#9DD5;
   // GBK_TO_UNICODE[42886] := 16#FA73;
   // GBK_TO_UNICODE[42887] := 16#9DD6;
   // GBK_TO_UNICODE[42888] := 16#FA74;
   // GBK_TO_UNICODE[42889] := 16#9DD7;
   // GBK_TO_UNICODE[42890] := 16#FA75;
   // GBK_TO_UNICODE[42891] := 16#9DD8;
   // GBK_TO_UNICODE[42892] := 16#FA76;
   // GBK_TO_UNICODE[42893] := 16#9DD9;
   // GBK_TO_UNICODE[42894] := 16#FA77;
   // GBK_TO_UNICODE[42895] := 16#9DDA;
   // GBK_TO_UNICODE[42896] := 16#FA78;
   // GBK_TO_UNICODE[42897] := 16#9DDB;
   // GBK_TO_UNICODE[42898] := 16#FA79;
   // GBK_TO_UNICODE[42899] := 16#9DDC;
   // GBK_TO_UNICODE[42900] := 16#FA7A;
   // GBK_TO_UNICODE[42901] := 16#9DDD;
   // GBK_TO_UNICODE[42902] := 16#FA7B;
   // GBK_TO_UNICODE[42903] := 16#9DDE;
   // GBK_TO_UNICODE[42904] := 16#FA7C;
   // GBK_TO_UNICODE[42905] := 16#9DDF;
   // GBK_TO_UNICODE[42906] := 16#FA7D;
   // GBK_TO_UNICODE[42907] := 16#9DE0;
   // GBK_TO_UNICODE[42908] := 16#FA7E;
   // GBK_TO_UNICODE[42909] := 16#9DE1;
   // GBK_TO_UNICODE[42910] := 16#FA80;
   // GBK_TO_UNICODE[42911] := 16#9DE2;
   // GBK_TO_UNICODE[42912] := 16#FA81;
   // GBK_TO_UNICODE[42913] := 16#9DE3;
   // GBK_TO_UNICODE[42914] := 16#FA82;
   // GBK_TO_UNICODE[42915] := 16#9DE4;
   // GBK_TO_UNICODE[42916] := 16#FA83;
   // GBK_TO_UNICODE[42917] := 16#9DE5;
   // GBK_TO_UNICODE[42918] := 16#FA84;
   // GBK_TO_UNICODE[42919] := 16#9DE6;
   // GBK_TO_UNICODE[42920] := 16#FA85;
   // GBK_TO_UNICODE[42921] := 16#9DE7;
   // GBK_TO_UNICODE[42922] := 16#FA86;
   // GBK_TO_UNICODE[42923] := 16#9DE8;
   // GBK_TO_UNICODE[42924] := 16#FA87;
   // GBK_TO_UNICODE[42925] := 16#9DE9;
   // GBK_TO_UNICODE[42926] := 16#FA88;
   // GBK_TO_UNICODE[42927] := 16#9DEA;
   // GBK_TO_UNICODE[42928] := 16#FA89;
   // GBK_TO_UNICODE[42929] := 16#9DEB;
   // GBK_TO_UNICODE[42930] := 16#FA8A;
   // GBK_TO_UNICODE[42931] := 16#9DEC;
   // GBK_TO_UNICODE[42932] := 16#FA8B;
   // GBK_TO_UNICODE[42933] := 16#9DED;
   // GBK_TO_UNICODE[42934] := 16#FA8C;
   // GBK_TO_UNICODE[42935] := 16#9DEE;
   // GBK_TO_UNICODE[42936] := 16#FA8D;
   // GBK_TO_UNICODE[42937] := 16#9DEF;
   // GBK_TO_UNICODE[42938] := 16#FA8E;
   // GBK_TO_UNICODE[42939] := 16#9DF0;
   // GBK_TO_UNICODE[42940] := 16#FA8F;
   // GBK_TO_UNICODE[42941] := 16#9DF1;
   // GBK_TO_UNICODE[42942] := 16#FA90;
   // GBK_TO_UNICODE[42943] := 16#9DF2;
   // GBK_TO_UNICODE[42944] := 16#FA91;
   // GBK_TO_UNICODE[42945] := 16#9DF3;
   // GBK_TO_UNICODE[42946] := 16#FA92;
   // GBK_TO_UNICODE[42947] := 16#9DF4;
   // GBK_TO_UNICODE[42948] := 16#FA93;
   // GBK_TO_UNICODE[42949] := 16#9DF5;
   // GBK_TO_UNICODE[42950] := 16#FA94;
   // GBK_TO_UNICODE[42951] := 16#9DF6;
   // GBK_TO_UNICODE[42952] := 16#FA95;
   // GBK_TO_UNICODE[42953] := 16#9DF7;
   // GBK_TO_UNICODE[42954] := 16#FA96;
   // GBK_TO_UNICODE[42955] := 16#9DF8;
   // GBK_TO_UNICODE[42956] := 16#FA97;
   // GBK_TO_UNICODE[42957] := 16#9DF9;
   // GBK_TO_UNICODE[42958] := 16#FA98;
   // GBK_TO_UNICODE[42959] := 16#9DFA;
   // GBK_TO_UNICODE[42960] := 16#FA99;
   // GBK_TO_UNICODE[42961] := 16#9DFB;
   // GBK_TO_UNICODE[42962] := 16#FA9A;
   // GBK_TO_UNICODE[42963] := 16#9DFC;
   // GBK_TO_UNICODE[42964] := 16#FA9B;
   // GBK_TO_UNICODE[42965] := 16#9DFD;
   // GBK_TO_UNICODE[42966] := 16#FA9C;
   // GBK_TO_UNICODE[42967] := 16#9DFE;
   // GBK_TO_UNICODE[42968] := 16#FA9D;
   // GBK_TO_UNICODE[42969] := 16#9DFF;
   // GBK_TO_UNICODE[42970] := 16#FA9E;
   // GBK_TO_UNICODE[42971] := 16#9E00;
   // GBK_TO_UNICODE[42972] := 16#FA9F;
   // GBK_TO_UNICODE[42973] := 16#9E01;
   // GBK_TO_UNICODE[42974] := 16#FAA0;
   // GBK_TO_UNICODE[42975] := 16#9E02;
   // GBK_TO_UNICODE[42976] := 16#FB40;
   // GBK_TO_UNICODE[42977] := 16#9E03;
   // GBK_TO_UNICODE[42978] := 16#FB41;
   // GBK_TO_UNICODE[42979] := 16#9E04;
   // GBK_TO_UNICODE[42980] := 16#FB42;
   // GBK_TO_UNICODE[42981] := 16#9E05;
   // GBK_TO_UNICODE[42982] := 16#FB43;
   // GBK_TO_UNICODE[42983] := 16#9E06;
   // GBK_TO_UNICODE[42984] := 16#FB44;
   // GBK_TO_UNICODE[42985] := 16#9E07;
   // GBK_TO_UNICODE[42986] := 16#FB45;
   // GBK_TO_UNICODE[42987] := 16#9E08;
   // GBK_TO_UNICODE[42988] := 16#FB46;
   // GBK_TO_UNICODE[42989] := 16#9E09;
   // GBK_TO_UNICODE[42990] := 16#FB47;
   // GBK_TO_UNICODE[42991] := 16#9E0A;
   // GBK_TO_UNICODE[42992] := 16#FB48;
   // GBK_TO_UNICODE[42993] := 16#9E0B;
   // GBK_TO_UNICODE[42994] := 16#FB49;
   // GBK_TO_UNICODE[42995] := 16#9E0C;
   // GBK_TO_UNICODE[42996] := 16#FB4A;
   // GBK_TO_UNICODE[42997] := 16#9E0D;
   // GBK_TO_UNICODE[42998] := 16#FB4B;
   // GBK_TO_UNICODE[42999] := 16#9E0E;
   // GBK_TO_UNICODE[43000] := 16#FB4C;
   // GBK_TO_UNICODE[43001] := 16#9E0F;
   // GBK_TO_UNICODE[43002] := 16#FB4D;
   // GBK_TO_UNICODE[43003] := 16#9E10;
   // GBK_TO_UNICODE[43004] := 16#FB4E;
   // GBK_TO_UNICODE[43005] := 16#9E11;
   // GBK_TO_UNICODE[43006] := 16#FB4F;
   // GBK_TO_UNICODE[43007] := 16#9E12;
   // GBK_TO_UNICODE[43008] := 16#FB50;
   // GBK_TO_UNICODE[43009] := 16#9E13;
   // GBK_TO_UNICODE[43010] := 16#FB51;
   // GBK_TO_UNICODE[43011] := 16#9E14;
   // GBK_TO_UNICODE[43012] := 16#FB52;
   // GBK_TO_UNICODE[43013] := 16#9E15;
   // GBK_TO_UNICODE[43014] := 16#FB53;
   // GBK_TO_UNICODE[43015] := 16#9E16;
   // GBK_TO_UNICODE[43016] := 16#FB54;
   // GBK_TO_UNICODE[43017] := 16#9E17;
   // GBK_TO_UNICODE[43018] := 16#FB55;
   // GBK_TO_UNICODE[43019] := 16#9E18;
   // GBK_TO_UNICODE[43020] := 16#FB56;
   // GBK_TO_UNICODE[43021] := 16#9E19;
   // GBK_TO_UNICODE[43022] := 16#FB57;
   // GBK_TO_UNICODE[43023] := 16#9E1A;
   // GBK_TO_UNICODE[43024] := 16#FB58;
   // GBK_TO_UNICODE[43025] := 16#9E1B;
   // GBK_TO_UNICODE[43026] := 16#FB59;
   // GBK_TO_UNICODE[43027] := 16#9E1C;
   // GBK_TO_UNICODE[43028] := 16#FB5A;
   // GBK_TO_UNICODE[43029] := 16#9E1D;
   // GBK_TO_UNICODE[43030] := 16#FB5B;
   // GBK_TO_UNICODE[43031] := 16#9E1E;
   // GBK_TO_UNICODE[43032] := 16#FB5C;
   // GBK_TO_UNICODE[43033] := 16#9E24;
   // GBK_TO_UNICODE[43034] := 16#FB5D;
   // GBK_TO_UNICODE[43035] := 16#9E27;
   // GBK_TO_UNICODE[43036] := 16#FB5E;
   // GBK_TO_UNICODE[43037] := 16#9E2E;
   // GBK_TO_UNICODE[43038] := 16#FB5F;
   // GBK_TO_UNICODE[43039] := 16#9E30;
   // GBK_TO_UNICODE[43040] := 16#FB60;
   // GBK_TO_UNICODE[43041] := 16#9E34;
   // GBK_TO_UNICODE[43042] := 16#FB61;
   // GBK_TO_UNICODE[43043] := 16#9E3B;
   // GBK_TO_UNICODE[43044] := 16#FB62;
   // GBK_TO_UNICODE[43045] := 16#9E3C;
   // GBK_TO_UNICODE[43046] := 16#FB63;
   // GBK_TO_UNICODE[43047] := 16#9E40;
   // GBK_TO_UNICODE[43048] := 16#FB64;
   // GBK_TO_UNICODE[43049] := 16#9E4D;
   // GBK_TO_UNICODE[43050] := 16#FB65;
   // GBK_TO_UNICODE[43051] := 16#9E50;
   // GBK_TO_UNICODE[43052] := 16#FB66;
   // GBK_TO_UNICODE[43053] := 16#9E52;
   // GBK_TO_UNICODE[43054] := 16#FB67;
   // GBK_TO_UNICODE[43055] := 16#9E53;
   // GBK_TO_UNICODE[43056] := 16#FB68;
   // GBK_TO_UNICODE[43057] := 16#9E54;
   // GBK_TO_UNICODE[43058] := 16#FB69;
   // GBK_TO_UNICODE[43059] := 16#9E56;
   // GBK_TO_UNICODE[43060] := 16#FB6A;
   // GBK_TO_UNICODE[43061] := 16#9E59;
   // GBK_TO_UNICODE[43062] := 16#FB6B;
   // GBK_TO_UNICODE[43063] := 16#9E5D;
   // GBK_TO_UNICODE[43064] := 16#FB6C;
   // GBK_TO_UNICODE[43065] := 16#9E5F;
   // GBK_TO_UNICODE[43066] := 16#FB6D;
   // GBK_TO_UNICODE[43067] := 16#9E60;
   // GBK_TO_UNICODE[43068] := 16#FB6E;
   // GBK_TO_UNICODE[43069] := 16#9E61;
   // GBK_TO_UNICODE[43070] := 16#FB6F;
   // GBK_TO_UNICODE[43071] := 16#9E62;
   // GBK_TO_UNICODE[43072] := 16#FB70;
   // GBK_TO_UNICODE[43073] := 16#9E65;
   // GBK_TO_UNICODE[43074] := 16#FB71;
   // GBK_TO_UNICODE[43075] := 16#9E6E;
   // GBK_TO_UNICODE[43076] := 16#FB72;
   // GBK_TO_UNICODE[43077] := 16#9E6F;
   // GBK_TO_UNICODE[43078] := 16#FB73;
   // GBK_TO_UNICODE[43079] := 16#9E72;
   // GBK_TO_UNICODE[43080] := 16#FB74;
   // GBK_TO_UNICODE[43081] := 16#9E74;
   // GBK_TO_UNICODE[43082] := 16#FB75;
   // GBK_TO_UNICODE[43083] := 16#9E75;
   // GBK_TO_UNICODE[43084] := 16#FB76;
   // GBK_TO_UNICODE[43085] := 16#9E76;
   // GBK_TO_UNICODE[43086] := 16#FB77;
   // GBK_TO_UNICODE[43087] := 16#9E77;
   // GBK_TO_UNICODE[43088] := 16#FB78;
   // GBK_TO_UNICODE[43089] := 16#9E78;
   // GBK_TO_UNICODE[43090] := 16#FB79;
   // GBK_TO_UNICODE[43091] := 16#9E79;
   // GBK_TO_UNICODE[43092] := 16#FB7A;
   // GBK_TO_UNICODE[43093] := 16#9E7A;
   // GBK_TO_UNICODE[43094] := 16#FB7B;
   // GBK_TO_UNICODE[43095] := 16#9E7B;
   // GBK_TO_UNICODE[43096] := 16#FB7C;
   // GBK_TO_UNICODE[43097] := 16#9E7C;
   // GBK_TO_UNICODE[43098] := 16#FB7D;
   // GBK_TO_UNICODE[43099] := 16#9E7D;
   // GBK_TO_UNICODE[43100] := 16#FB7E;
   // GBK_TO_UNICODE[43101] := 16#9E80;
   // GBK_TO_UNICODE[43102] := 16#FB80;
   // GBK_TO_UNICODE[43103] := 16#9E81;
   // GBK_TO_UNICODE[43104] := 16#FB81;
   // GBK_TO_UNICODE[43105] := 16#9E83;
   // GBK_TO_UNICODE[43106] := 16#FB82;
   // GBK_TO_UNICODE[43107] := 16#9E84;
   // GBK_TO_UNICODE[43108] := 16#FB83;
   // GBK_TO_UNICODE[43109] := 16#9E85;
   // GBK_TO_UNICODE[43110] := 16#FB84;
   // GBK_TO_UNICODE[43111] := 16#9E86;
   // GBK_TO_UNICODE[43112] := 16#FB85;
   // GBK_TO_UNICODE[43113] := 16#9E89;
   // GBK_TO_UNICODE[43114] := 16#FB86;
   // GBK_TO_UNICODE[43115] := 16#9E8A;
   // GBK_TO_UNICODE[43116] := 16#FB87;
   // GBK_TO_UNICODE[43117] := 16#9E8C;
   // GBK_TO_UNICODE[43118] := 16#FB88;
   // GBK_TO_UNICODE[43119] := 16#9E8D;
   // GBK_TO_UNICODE[43120] := 16#FB89;
   // GBK_TO_UNICODE[43121] := 16#9E8E;
   // GBK_TO_UNICODE[43122] := 16#FB8A;
   // GBK_TO_UNICODE[43123] := 16#9E8F;
   // GBK_TO_UNICODE[43124] := 16#FB8B;
   // GBK_TO_UNICODE[43125] := 16#9E90;
   // GBK_TO_UNICODE[43126] := 16#FB8C;
   // GBK_TO_UNICODE[43127] := 16#9E91;
   // GBK_TO_UNICODE[43128] := 16#FB8D;
   // GBK_TO_UNICODE[43129] := 16#9E94;
   // GBK_TO_UNICODE[43130] := 16#FB8E;
   // GBK_TO_UNICODE[43131] := 16#9E95;
   // GBK_TO_UNICODE[43132] := 16#FB8F;
   // GBK_TO_UNICODE[43133] := 16#9E96;
   // GBK_TO_UNICODE[43134] := 16#FB90;
   // GBK_TO_UNICODE[43135] := 16#9E97;
   // GBK_TO_UNICODE[43136] := 16#FB91;
   // GBK_TO_UNICODE[43137] := 16#9E98;
   // GBK_TO_UNICODE[43138] := 16#FB92;
   // GBK_TO_UNICODE[43139] := 16#9E99;
   // GBK_TO_UNICODE[43140] := 16#FB93;
   // GBK_TO_UNICODE[43141] := 16#9E9A;
   // GBK_TO_UNICODE[43142] := 16#FB94;
   // GBK_TO_UNICODE[43143] := 16#9E9B;
   // GBK_TO_UNICODE[43144] := 16#FB95;
   // GBK_TO_UNICODE[43145] := 16#9E9C;
   // GBK_TO_UNICODE[43146] := 16#FB96;
   // GBK_TO_UNICODE[43147] := 16#9E9E;
   // GBK_TO_UNICODE[43148] := 16#FB97;
   // GBK_TO_UNICODE[43149] := 16#9EA0;
   // GBK_TO_UNICODE[43150] := 16#FB98;
   // GBK_TO_UNICODE[43151] := 16#9EA1;
   // GBK_TO_UNICODE[43152] := 16#FB99;
   // GBK_TO_UNICODE[43153] := 16#9EA2;
   // GBK_TO_UNICODE[43154] := 16#FB9A;
   // GBK_TO_UNICODE[43155] := 16#9EA3;
   // GBK_TO_UNICODE[43156] := 16#FB9B;
   // GBK_TO_UNICODE[43157] := 16#9EA4;
   // GBK_TO_UNICODE[43158] := 16#FB9C;
   // GBK_TO_UNICODE[43159] := 16#9EA5;
   // GBK_TO_UNICODE[43160] := 16#FB9D;
   // GBK_TO_UNICODE[43161] := 16#9EA7;
   // GBK_TO_UNICODE[43162] := 16#FB9E;
   // GBK_TO_UNICODE[43163] := 16#9EA8;
   // GBK_TO_UNICODE[43164] := 16#FB9F;
   // GBK_TO_UNICODE[43165] := 16#9EA9;
   // GBK_TO_UNICODE[43166] := 16#FBA0;
   // GBK_TO_UNICODE[43167] := 16#9EAA;
   // GBK_TO_UNICODE[43168] := 16#FC40;
   // GBK_TO_UNICODE[43169] := 16#9EAB;
   // GBK_TO_UNICODE[43170] := 16#FC41;
   // GBK_TO_UNICODE[43171] := 16#9EAC;
   // GBK_TO_UNICODE[43172] := 16#FC42;
   // GBK_TO_UNICODE[43173] := 16#9EAD;
   // GBK_TO_UNICODE[43174] := 16#FC43;
   // GBK_TO_UNICODE[43175] := 16#9EAE;
   // GBK_TO_UNICODE[43176] := 16#FC44;
   // GBK_TO_UNICODE[43177] := 16#9EAF;
   // GBK_TO_UNICODE[43178] := 16#FC45;
   // GBK_TO_UNICODE[43179] := 16#9EB0;
   // GBK_TO_UNICODE[43180] := 16#FC46;
   // GBK_TO_UNICODE[43181] := 16#9EB1;
   // GBK_TO_UNICODE[43182] := 16#FC47;
   // GBK_TO_UNICODE[43183] := 16#9EB2;
   // GBK_TO_UNICODE[43184] := 16#FC48;
   // GBK_TO_UNICODE[43185] := 16#9EB3;
   // GBK_TO_UNICODE[43186] := 16#FC49;
   // GBK_TO_UNICODE[43187] := 16#9EB5;
   // GBK_TO_UNICODE[43188] := 16#FC4A;
   // GBK_TO_UNICODE[43189] := 16#9EB6;
   // GBK_TO_UNICODE[43190] := 16#FC4B;
   // GBK_TO_UNICODE[43191] := 16#9EB7;
   // GBK_TO_UNICODE[43192] := 16#FC4C;
   // GBK_TO_UNICODE[43193] := 16#9EB9;
   // GBK_TO_UNICODE[43194] := 16#FC4D;
   // GBK_TO_UNICODE[43195] := 16#9EBA;
   // GBK_TO_UNICODE[43196] := 16#FC4E;
   // GBK_TO_UNICODE[43197] := 16#9EBC;
   // GBK_TO_UNICODE[43198] := 16#FC4F;
   // GBK_TO_UNICODE[43199] := 16#9EBF;
   // GBK_TO_UNICODE[43200] := 16#FC50;
   // GBK_TO_UNICODE[43201] := 16#9EC0;
   // GBK_TO_UNICODE[43202] := 16#FC51;
   // GBK_TO_UNICODE[43203] := 16#9EC1;
   // GBK_TO_UNICODE[43204] := 16#FC52;
   // GBK_TO_UNICODE[43205] := 16#9EC2;
   // GBK_TO_UNICODE[43206] := 16#FC53;
   // GBK_TO_UNICODE[43207] := 16#9EC3;
   // GBK_TO_UNICODE[43208] := 16#FC54;
   // GBK_TO_UNICODE[43209] := 16#9EC5;
   // GBK_TO_UNICODE[43210] := 16#FC55;
   // GBK_TO_UNICODE[43211] := 16#9EC6;
   // GBK_TO_UNICODE[43212] := 16#FC56;
   // GBK_TO_UNICODE[43213] := 16#9EC7;
   // GBK_TO_UNICODE[43214] := 16#FC57;
   // GBK_TO_UNICODE[43215] := 16#9EC8;
   // GBK_TO_UNICODE[43216] := 16#FC58;
   // GBK_TO_UNICODE[43217] := 16#9ECA;
   // GBK_TO_UNICODE[43218] := 16#FC59;
   // GBK_TO_UNICODE[43219] := 16#9ECB;
   // GBK_TO_UNICODE[43220] := 16#FC5A;
   // GBK_TO_UNICODE[43221] := 16#9ECC;
   // GBK_TO_UNICODE[43222] := 16#FC5B;
   // GBK_TO_UNICODE[43223] := 16#9ED0;
   // GBK_TO_UNICODE[43224] := 16#FC5C;
   // GBK_TO_UNICODE[43225] := 16#9ED2;
   // GBK_TO_UNICODE[43226] := 16#FC5D;
   // GBK_TO_UNICODE[43227] := 16#9ED3;
   // GBK_TO_UNICODE[43228] := 16#FC5E;
   // GBK_TO_UNICODE[43229] := 16#9ED5;
   // GBK_TO_UNICODE[43230] := 16#FC5F;
   // GBK_TO_UNICODE[43231] := 16#9ED6;
   // GBK_TO_UNICODE[43232] := 16#FC60;
   // GBK_TO_UNICODE[43233] := 16#9ED7;
   // GBK_TO_UNICODE[43234] := 16#FC61;
   // GBK_TO_UNICODE[43235] := 16#9ED9;
   // GBK_TO_UNICODE[43236] := 16#FC62;
   // GBK_TO_UNICODE[43237] := 16#9EDA;
   // GBK_TO_UNICODE[43238] := 16#FC63;
   // GBK_TO_UNICODE[43239] := 16#9EDE;
   // GBK_TO_UNICODE[43240] := 16#FC64;
   // GBK_TO_UNICODE[43241] := 16#9EE1;
   // GBK_TO_UNICODE[43242] := 16#FC65;
   // GBK_TO_UNICODE[43243] := 16#9EE3;
   // GBK_TO_UNICODE[43244] := 16#FC66;
   // GBK_TO_UNICODE[43245] := 16#9EE4;
   // GBK_TO_UNICODE[43246] := 16#FC67;
   // GBK_TO_UNICODE[43247] := 16#9EE6;
   // GBK_TO_UNICODE[43248] := 16#FC68;
   // GBK_TO_UNICODE[43249] := 16#9EE8;
   // GBK_TO_UNICODE[43250] := 16#FC69;
   // GBK_TO_UNICODE[43251] := 16#9EEB;
   // GBK_TO_UNICODE[43252] := 16#FC6A;
   // GBK_TO_UNICODE[43253] := 16#9EEC;
   // GBK_TO_UNICODE[43254] := 16#FC6B;
   // GBK_TO_UNICODE[43255] := 16#9EED;
   // GBK_TO_UNICODE[43256] := 16#FC6C;
   // GBK_TO_UNICODE[43257] := 16#9EEE;
   // GBK_TO_UNICODE[43258] := 16#FC6D;
   // GBK_TO_UNICODE[43259] := 16#9EF0;
   // GBK_TO_UNICODE[43260] := 16#FC6E;
   // GBK_TO_UNICODE[43261] := 16#9EF1;
   // GBK_TO_UNICODE[43262] := 16#FC6F;
   // GBK_TO_UNICODE[43263] := 16#9EF2;
   // GBK_TO_UNICODE[43264] := 16#FC70;
   // GBK_TO_UNICODE[43265] := 16#9EF3;
   // GBK_TO_UNICODE[43266] := 16#FC71;
   // GBK_TO_UNICODE[43267] := 16#9EF4;
   // GBK_TO_UNICODE[43268] := 16#FC72;
   // GBK_TO_UNICODE[43269] := 16#9EF5;
   // GBK_TO_UNICODE[43270] := 16#FC73;
   // GBK_TO_UNICODE[43271] := 16#9EF6;
   // GBK_TO_UNICODE[43272] := 16#FC74;
   // GBK_TO_UNICODE[43273] := 16#9EF7;
   // GBK_TO_UNICODE[43274] := 16#FC75;
   // GBK_TO_UNICODE[43275] := 16#9EF8;
   // GBK_TO_UNICODE[43276] := 16#FC76;
   // GBK_TO_UNICODE[43277] := 16#9EFA;
   // GBK_TO_UNICODE[43278] := 16#FC77;
   // GBK_TO_UNICODE[43279] := 16#9EFD;
   // GBK_TO_UNICODE[43280] := 16#FC78;
   // GBK_TO_UNICODE[43281] := 16#9EFF;
   // GBK_TO_UNICODE[43282] := 16#FC79;
   // GBK_TO_UNICODE[43283] := 16#9F00;
   // GBK_TO_UNICODE[43284] := 16#FC7A;
   // GBK_TO_UNICODE[43285] := 16#9F01;
   // GBK_TO_UNICODE[43286] := 16#FC7B;
   // GBK_TO_UNICODE[43287] := 16#9F02;
   // GBK_TO_UNICODE[43288] := 16#FC7C;
   // GBK_TO_UNICODE[43289] := 16#9F03;
   // GBK_TO_UNICODE[43290] := 16#FC7D;
   // GBK_TO_UNICODE[43291] := 16#9F04;
   // GBK_TO_UNICODE[43292] := 16#FC7E;
   // GBK_TO_UNICODE[43293] := 16#9F05;
   // GBK_TO_UNICODE[43294] := 16#FC80;
   // GBK_TO_UNICODE[43295] := 16#9F06;
   // GBK_TO_UNICODE[43296] := 16#FC81;
   // GBK_TO_UNICODE[43297] := 16#9F07;
   // GBK_TO_UNICODE[43298] := 16#FC82;
   // GBK_TO_UNICODE[43299] := 16#9F08;
   // GBK_TO_UNICODE[43300] := 16#FC83;
   // GBK_TO_UNICODE[43301] := 16#9F09;
   // GBK_TO_UNICODE[43302] := 16#FC84;
   // GBK_TO_UNICODE[43303] := 16#9F0A;
   // GBK_TO_UNICODE[43304] := 16#FC85;
   // GBK_TO_UNICODE[43305] := 16#9F0C;
   // GBK_TO_UNICODE[43306] := 16#FC86;
   // GBK_TO_UNICODE[43307] := 16#9F0F;
   // GBK_TO_UNICODE[43308] := 16#FC87;
   // GBK_TO_UNICODE[43309] := 16#9F11;
   // GBK_TO_UNICODE[43310] := 16#FC88;
   // GBK_TO_UNICODE[43311] := 16#9F12;
   // GBK_TO_UNICODE[43312] := 16#FC89;
   // GBK_TO_UNICODE[43313] := 16#9F14;
   // GBK_TO_UNICODE[43314] := 16#FC8A;
   // GBK_TO_UNICODE[43315] := 16#9F15;
   // GBK_TO_UNICODE[43316] := 16#FC8B;
   // GBK_TO_UNICODE[43317] := 16#9F16;
   // GBK_TO_UNICODE[43318] := 16#FC8C;
   // GBK_TO_UNICODE[43319] := 16#9F18;
   // GBK_TO_UNICODE[43320] := 16#FC8D;
   // GBK_TO_UNICODE[43321] := 16#9F1A;
   // GBK_TO_UNICODE[43322] := 16#FC8E;
   // GBK_TO_UNICODE[43323] := 16#9F1B;
   // GBK_TO_UNICODE[43324] := 16#FC8F;
   // GBK_TO_UNICODE[43325] := 16#9F1C;
   // GBK_TO_UNICODE[43326] := 16#FC90;
   // GBK_TO_UNICODE[43327] := 16#9F1D;
   // GBK_TO_UNICODE[43328] := 16#FC91;
   // GBK_TO_UNICODE[43329] := 16#9F1E;
   // GBK_TO_UNICODE[43330] := 16#FC92;
   // GBK_TO_UNICODE[43331] := 16#9F1F;
   // GBK_TO_UNICODE[43332] := 16#FC93;
   // GBK_TO_UNICODE[43333] := 16#9F21;
   // GBK_TO_UNICODE[43334] := 16#FC94;
   // GBK_TO_UNICODE[43335] := 16#9F23;
   // GBK_TO_UNICODE[43336] := 16#FC95;
   // GBK_TO_UNICODE[43337] := 16#9F24;
   // GBK_TO_UNICODE[43338] := 16#FC96;
   // GBK_TO_UNICODE[43339] := 16#9F25;
   // GBK_TO_UNICODE[43340] := 16#FC97;
   // GBK_TO_UNICODE[43341] := 16#9F26;
   // GBK_TO_UNICODE[43342] := 16#FC98;
   // GBK_TO_UNICODE[43343] := 16#9F27;
   // GBK_TO_UNICODE[43344] := 16#FC99;
   // GBK_TO_UNICODE[43345] := 16#9F28;
   // GBK_TO_UNICODE[43346] := 16#FC9A;
   // GBK_TO_UNICODE[43347] := 16#9F29;
   // GBK_TO_UNICODE[43348] := 16#FC9B;
   // GBK_TO_UNICODE[43349] := 16#9F2A;
   // GBK_TO_UNICODE[43350] := 16#FC9C;
   // GBK_TO_UNICODE[43351] := 16#9F2B;
   // GBK_TO_UNICODE[43352] := 16#FC9D;
   // GBK_TO_UNICODE[43353] := 16#9F2D;
   // GBK_TO_UNICODE[43354] := 16#FC9E;
   // GBK_TO_UNICODE[43355] := 16#9F2E;
   // GBK_TO_UNICODE[43356] := 16#FC9F;
   // GBK_TO_UNICODE[43357] := 16#9F30;
   // GBK_TO_UNICODE[43358] := 16#FCA0;
   // GBK_TO_UNICODE[43359] := 16#9F31;
   // GBK_TO_UNICODE[43360] := 16#FD40;
   // GBK_TO_UNICODE[43361] := 16#9F32;
   // GBK_TO_UNICODE[43362] := 16#FD41;
   // GBK_TO_UNICODE[43363] := 16#9F33;
   // GBK_TO_UNICODE[43364] := 16#FD42;
   // GBK_TO_UNICODE[43365] := 16#9F34;
   // GBK_TO_UNICODE[43366] := 16#FD43;
   // GBK_TO_UNICODE[43367] := 16#9F35;
   // GBK_TO_UNICODE[43368] := 16#FD44;
   // GBK_TO_UNICODE[43369] := 16#9F36;
   // GBK_TO_UNICODE[43370] := 16#FD45;
   // GBK_TO_UNICODE[43371] := 16#9F38;
   // GBK_TO_UNICODE[43372] := 16#FD46;
   // GBK_TO_UNICODE[43373] := 16#9F3A;
   // GBK_TO_UNICODE[43374] := 16#FD47;
   // GBK_TO_UNICODE[43375] := 16#9F3C;
   // GBK_TO_UNICODE[43376] := 16#FD48;
   // GBK_TO_UNICODE[43377] := 16#9F3F;
   // GBK_TO_UNICODE[43378] := 16#FD49;
   // GBK_TO_UNICODE[43379] := 16#9F40;
   // GBK_TO_UNICODE[43380] := 16#FD4A;
   // GBK_TO_UNICODE[43381] := 16#9F41;
   // GBK_TO_UNICODE[43382] := 16#FD4B;
   // GBK_TO_UNICODE[43383] := 16#9F42;
   // GBK_TO_UNICODE[43384] := 16#FD4C;
   // GBK_TO_UNICODE[43385] := 16#9F43;
   // GBK_TO_UNICODE[43386] := 16#FD4D;
   // GBK_TO_UNICODE[43387] := 16#9F45;
   // GBK_TO_UNICODE[43388] := 16#FD4E;
   // GBK_TO_UNICODE[43389] := 16#9F46;
   // GBK_TO_UNICODE[43390] := 16#FD4F;
   // GBK_TO_UNICODE[43391] := 16#9F47;
   // GBK_TO_UNICODE[43392] := 16#FD50;
   // GBK_TO_UNICODE[43393] := 16#9F48;
   // GBK_TO_UNICODE[43394] := 16#FD51;
   // GBK_TO_UNICODE[43395] := 16#9F49;
   // GBK_TO_UNICODE[43396] := 16#FD52;
   // GBK_TO_UNICODE[43397] := 16#9F4A;
   // GBK_TO_UNICODE[43398] := 16#FD53;
   // GBK_TO_UNICODE[43399] := 16#9F4B;
   // GBK_TO_UNICODE[43400] := 16#FD54;
   // GBK_TO_UNICODE[43401] := 16#9F4C;
   // GBK_TO_UNICODE[43402] := 16#FD55;
   // GBK_TO_UNICODE[43403] := 16#9F4D;
   // GBK_TO_UNICODE[43404] := 16#FD56;
   // GBK_TO_UNICODE[43405] := 16#9F4E;
   // GBK_TO_UNICODE[43406] := 16#FD57;
   // GBK_TO_UNICODE[43407] := 16#9F4F;
   // GBK_TO_UNICODE[43408] := 16#FD58;
   // GBK_TO_UNICODE[43409] := 16#9F52;
   // GBK_TO_UNICODE[43410] := 16#FD59;
   // GBK_TO_UNICODE[43411] := 16#9F53;
   // GBK_TO_UNICODE[43412] := 16#FD5A;
   // GBK_TO_UNICODE[43413] := 16#9F54;
   // GBK_TO_UNICODE[43414] := 16#FD5B;
   // GBK_TO_UNICODE[43415] := 16#9F55;
   // GBK_TO_UNICODE[43416] := 16#FD5C;
   // GBK_TO_UNICODE[43417] := 16#9F56;
   // GBK_TO_UNICODE[43418] := 16#FD5D;
   // GBK_TO_UNICODE[43419] := 16#9F57;
   // GBK_TO_UNICODE[43420] := 16#FD5E;
   // GBK_TO_UNICODE[43421] := 16#9F58;
   // GBK_TO_UNICODE[43422] := 16#FD5F;
   // GBK_TO_UNICODE[43423] := 16#9F59;
   // GBK_TO_UNICODE[43424] := 16#FD60;
   // GBK_TO_UNICODE[43425] := 16#9F5A;
   // GBK_TO_UNICODE[43426] := 16#FD61;
   // GBK_TO_UNICODE[43427] := 16#9F5B;
   // GBK_TO_UNICODE[43428] := 16#FD62;
   // GBK_TO_UNICODE[43429] := 16#9F5C;
   // GBK_TO_UNICODE[43430] := 16#FD63;
   // GBK_TO_UNICODE[43431] := 16#9F5D;
   // GBK_TO_UNICODE[43432] := 16#FD64;
   // GBK_TO_UNICODE[43433] := 16#9F5E;
   // GBK_TO_UNICODE[43434] := 16#FD65;
   // GBK_TO_UNICODE[43435] := 16#9F5F;
   // GBK_TO_UNICODE[43436] := 16#FD66;
   // GBK_TO_UNICODE[43437] := 16#9F60;
   // GBK_TO_UNICODE[43438] := 16#FD67;
   // GBK_TO_UNICODE[43439] := 16#9F61;
   // GBK_TO_UNICODE[43440] := 16#FD68;
   // GBK_TO_UNICODE[43441] := 16#9F62;
   // GBK_TO_UNICODE[43442] := 16#FD69;
   // GBK_TO_UNICODE[43443] := 16#9F63;
   // GBK_TO_UNICODE[43444] := 16#FD6A;
   // GBK_TO_UNICODE[43445] := 16#9F64;
   // GBK_TO_UNICODE[43446] := 16#FD6B;
   // GBK_TO_UNICODE[43447] := 16#9F65;
   // GBK_TO_UNICODE[43448] := 16#FD6C;
   // GBK_TO_UNICODE[43449] := 16#9F66;
   // GBK_TO_UNICODE[43450] := 16#FD6D;
   // GBK_TO_UNICODE[43451] := 16#9F67;
   // GBK_TO_UNICODE[43452] := 16#FD6E;
   // GBK_TO_UNICODE[43453] := 16#9F68;
   // GBK_TO_UNICODE[43454] := 16#FD6F;
   // GBK_TO_UNICODE[43455] := 16#9F69;
   // GBK_TO_UNICODE[43456] := 16#FD70;
   // GBK_TO_UNICODE[43457] := 16#9F6A;
   // GBK_TO_UNICODE[43458] := 16#FD71;
   // GBK_TO_UNICODE[43459] := 16#9F6B;
   // GBK_TO_UNICODE[43460] := 16#FD72;
   // GBK_TO_UNICODE[43461] := 16#9F6C;
   // GBK_TO_UNICODE[43462] := 16#FD73;
   // GBK_TO_UNICODE[43463] := 16#9F6D;
   // GBK_TO_UNICODE[43464] := 16#FD74;
   // GBK_TO_UNICODE[43465] := 16#9F6E;
   // GBK_TO_UNICODE[43466] := 16#FD75;
   // GBK_TO_UNICODE[43467] := 16#9F6F;
   // GBK_TO_UNICODE[43468] := 16#FD76;
   // GBK_TO_UNICODE[43469] := 16#9F70;
   // GBK_TO_UNICODE[43470] := 16#FD77;
   // GBK_TO_UNICODE[43471] := 16#9F71;
   // GBK_TO_UNICODE[43472] := 16#FD78;
   // GBK_TO_UNICODE[43473] := 16#9F72;
   // GBK_TO_UNICODE[43474] := 16#FD79;
   // GBK_TO_UNICODE[43475] := 16#9F73;
   // GBK_TO_UNICODE[43476] := 16#FD7A;
   // GBK_TO_UNICODE[43477] := 16#9F74;
   // GBK_TO_UNICODE[43478] := 16#FD7B;
   // GBK_TO_UNICODE[43479] := 16#9F75;
   // GBK_TO_UNICODE[43480] := 16#FD7C;
   // GBK_TO_UNICODE[43481] := 16#9F76;
   // GBK_TO_UNICODE[43482] := 16#FD7D;
   // GBK_TO_UNICODE[43483] := 16#9F77;
   // GBK_TO_UNICODE[43484] := 16#FD7E;
   // GBK_TO_UNICODE[43485] := 16#9F78;
   // GBK_TO_UNICODE[43486] := 16#FD80;
   // GBK_TO_UNICODE[43487] := 16#9F79;
   // GBK_TO_UNICODE[43488] := 16#FD81;
   // GBK_TO_UNICODE[43489] := 16#9F7A;
   // GBK_TO_UNICODE[43490] := 16#FD82;
   // GBK_TO_UNICODE[43491] := 16#9F7B;
   // GBK_TO_UNICODE[43492] := 16#FD83;
   // GBK_TO_UNICODE[43493] := 16#9F7C;
   // GBK_TO_UNICODE[43494] := 16#FD84;
   // GBK_TO_UNICODE[43495] := 16#9F7D;
   // GBK_TO_UNICODE[43496] := 16#FD85;
   // GBK_TO_UNICODE[43497] := 16#9F7E;
   // GBK_TO_UNICODE[43498] := 16#FD86;
   // GBK_TO_UNICODE[43499] := 16#9F81;
   // GBK_TO_UNICODE[43500] := 16#FD87;
   // GBK_TO_UNICODE[43501] := 16#9F82;
   // GBK_TO_UNICODE[43502] := 16#FD88;
   // GBK_TO_UNICODE[43503] := 16#9F8D;
   // GBK_TO_UNICODE[43504] := 16#FD89;
   // GBK_TO_UNICODE[43505] := 16#9F8E;
   // GBK_TO_UNICODE[43506] := 16#FD8A;
   // GBK_TO_UNICODE[43507] := 16#9F8F;
   // GBK_TO_UNICODE[43508] := 16#FD8B;
   // GBK_TO_UNICODE[43509] := 16#9F90;
   // GBK_TO_UNICODE[43510] := 16#FD8C;
   // GBK_TO_UNICODE[43511] := 16#9F91;
   // GBK_TO_UNICODE[43512] := 16#FD8D;
   // GBK_TO_UNICODE[43513] := 16#9F92;
   // GBK_TO_UNICODE[43514] := 16#FD8E;
   // GBK_TO_UNICODE[43515] := 16#9F93;
   // GBK_TO_UNICODE[43516] := 16#FD8F;
   // GBK_TO_UNICODE[43517] := 16#9F94;
   // GBK_TO_UNICODE[43518] := 16#FD90;
   // GBK_TO_UNICODE[43519] := 16#9F95;
   // GBK_TO_UNICODE[43520] := 16#FD91;
   // GBK_TO_UNICODE[43521] := 16#9F96;
   // GBK_TO_UNICODE[43522] := 16#FD92;
   // GBK_TO_UNICODE[43523] := 16#9F97;
   // GBK_TO_UNICODE[43524] := 16#FD93;
   // GBK_TO_UNICODE[43525] := 16#9F98;
   // GBK_TO_UNICODE[43526] := 16#FD94;
   // GBK_TO_UNICODE[43527] := 16#9F9C;
   // GBK_TO_UNICODE[43528] := 16#FD95;
   // GBK_TO_UNICODE[43529] := 16#9F9D;
   // GBK_TO_UNICODE[43530] := 16#FD96;
   // GBK_TO_UNICODE[43531] := 16#9F9E;
   // GBK_TO_UNICODE[43532] := 16#FD97;
   // GBK_TO_UNICODE[43533] := 16#9FA1;
   // GBK_TO_UNICODE[43534] := 16#FD98;
   // GBK_TO_UNICODE[43535] := 16#9FA2;
   // GBK_TO_UNICODE[43536] := 16#FD99;
   // GBK_TO_UNICODE[43537] := 16#9FA3;
   // GBK_TO_UNICODE[43538] := 16#FD9A;
   // GBK_TO_UNICODE[43539] := 16#9FA4;
   // GBK_TO_UNICODE[43540] := 16#FD9B;
   // GBK_TO_UNICODE[43541] := 16#9FA5;
   // GBK_TO_UNICODE[43542] := 16#FD9C;
   // GBK_TO_UNICODE[43543] := 16#F92C;
   // GBK_TO_UNICODE[43544] := 16#FD9D;
   // GBK_TO_UNICODE[43545] := 16#F979;
   // GBK_TO_UNICODE[43546] := 16#FD9E;
   // GBK_TO_UNICODE[43547] := 16#F995;
   // GBK_TO_UNICODE[43548] := 16#FD9F;
   // GBK_TO_UNICODE[43549] := 16#F9E7;
   // GBK_TO_UNICODE[43550] := 16#FDA0;
   // GBK_TO_UNICODE[43551] := 16#F9F1;
   // GBK_TO_UNICODE[43552] := 16#FE40;
   // GBK_TO_UNICODE[43553] := 16#FA0C;
   // GBK_TO_UNICODE[43554] := 16#FE41;
   // GBK_TO_UNICODE[43555] := 16#FA0D;
   // GBK_TO_UNICODE[43556] := 16#FE42;
   // GBK_TO_UNICODE[43557] := 16#FA0E;
   // GBK_TO_UNICODE[43558] := 16#FE43;
   // GBK_TO_UNICODE[43559] := 16#FA0F;
   // GBK_TO_UNICODE[43560] := 16#FE44;
   // GBK_TO_UNICODE[43561] := 16#FA11;
   // GBK_TO_UNICODE[43562] := 16#FE45;
   // GBK_TO_UNICODE[43563] := 16#FA13;
   // GBK_TO_UNICODE[43564] := 16#FE46;
   // GBK_TO_UNICODE[43565] := 16#FA14;
   // GBK_TO_UNICODE[43566] := 16#FE47;
   // GBK_TO_UNICODE[43567] := 16#FA18;
   // GBK_TO_UNICODE[43568] := 16#FE48;
   // GBK_TO_UNICODE[43569] := 16#FA1F;
   // GBK_TO_UNICODE[43570] := 16#FE49;
   // GBK_TO_UNICODE[43571] := 16#FA20;
   // GBK_TO_UNICODE[43572] := 16#FE4A;
   // GBK_TO_UNICODE[43573] := 16#FA21;
   // GBK_TO_UNICODE[43574] := 16#FE4B;
   // GBK_TO_UNICODE[43575] := 16#FA23;
   // GBK_TO_UNICODE[43576] := 16#FE4C;
   // GBK_TO_UNICODE[43577] := 16#FA24;
   // GBK_TO_UNICODE[43578] := 16#FE4D;
   // GBK_TO_UNICODE[43579] := 16#FA27;
   // GBK_TO_UNICODE[43580] := 16#FE4E;
   // GBK_TO_UNICODE[43581] := 16#FA28;
   // GBK_TO_UNICODE[43582] := 16#FE4F;
   // GBK_TO_UNICODE[43583] := 16#FA29;
   // GBK_TO_UNICODE[43584] := 0;
   // GBK_TO_UNICODE[43585] := 0;
BEGIN
   IF #GBK < 16#0080 THEN
       #UNICODE := #GBK;
   ELSE
       #hi := 21796;
       #li := 0;
       FOR #j := 0 TO 16 BY 1 DO
           #i := #li + (#hi - #li) / 2;
           IF #GBK = #GBK_TO_UNICODE[#i * 2] THEN
               #UNICODE := #GBK_TO_UNICODE[#i * 2 + 1];
               EXIT;
           END_IF;
           IF #GBK > #GBK_TO_UNICODE[#i * 2] THEN
               #li := #i;
           ELSE
               #hi := #i;
           END_IF;
       END_FOR;
   END_IF;
END_FUNCTION_BLOCK

// ===== library: MasterCopy "UNI_TO_GB2" =====

// folder: FB/UNICODE_FB

